FUNCTION_BLOCK fb_debugData
VAR_INPUT
END_VAR
VAR_OUTPUT
END_VAR
VAR
	productID: INT;
END_VAR

productID := 0;


gvl_param.var_productInfo[productID].name 				:= '---ForDebug---';
gvl_param.var_productInfo[productID].num				:= productID;
gvl_param.var_productInfo[productID].bottomPocketQty 	:= 5;
gvl_param.var_productInfo[productID].vertivalPocketQty 	:= 3;
gvl_param.var_productInfo[productID].startCav 			:= 1;
gvl_param.var_productInfo[productID].cavQty 			:= 8;
gvl_param.var_productInfo[productID].gateLength_max 	:= 30000;
gvl_param.var_productInfo[productID].gateLength_min 	:= 15000;
gvl_param.var_productInfo[productID].pocketSumQty		:= 15;
gvl_param.var_productInfo[productID].autoVels.x.vel		:= 300;
gvl_param.var_productInfo[productID].autoVels.x.acc		:= 10000;
gvl_param.var_productInfo[productID].autoVels.x.dcc		:= 10000;
gvl_param.var_productInfo[productID].autoVels.y.vel		:= 150;
gvl_param.var_productInfo[productID].autoVels.y.acc		:= 10000;
gvl_param.var_productInfo[productID].autoVels.y.dcc		:= 10000;
gvl_param.var_productInfo[productID].autoVels.z.vel		:= 150;
gvl_param.var_productInfo[productID].autoVels.z.acc		:= 10000;
gvl_param.var_productInfo[productID].autoVels.z.dcc		:= 10000;
gvl_param.var_productInfo[productID].manaulVels.x.vel	:= 100;
gvl_param.var_productInfo[productID].manaulVels.y.vel	:= 50;
gvl_param.var_productInfo[productID].manaulVels.z.vel	:= 50;

gvl_param.var_productInfo[productID].teachPos.initial.x	:= 950;
gvl_param.var_productInfo[productID].teachPos.initial.y	:= 30;
gvl_param.var_productInfo[productID].teachPos.initial.z	:= 0;
gvl_param.var_productInfo[productID].teachPos.pickUp.x	:= 1250;
gvl_param.var_productInfo[productID].teachPos.pickUp.y	:= 30;
gvl_param.var_productInfo[productID].teachPos.pickUp.z	:= 10;
gvl_param.var_productInfo[productID].teachPos.remove.x	:= 1220;
gvl_param.var_productInfo[productID].teachPos.remove.y	:= 190;
gvl_param.var_productInfo[productID].teachPos.remove.z	:= 10;
//#1
gvl_param.var_productInfo[productID].teachPos.palletize.upperLower[1].cav[1].Pos[1].x := 1007;
gvl_param.var_productInfo[productID].teachPos.palletize.upperLower[1].cav[1].Pos[1].y := 54;
gvl_param.var_productInfo[productID].teachPos.palletize.upperLower[1].cav[1].Pos[1].z := 15;
gvl_param.var_productInfo[productID].teachPos.palletize.upperLower[1].cav[1].Pos[2].x := 1084;
gvl_param.var_productInfo[productID].teachPos.palletize.upperLower[1].cav[1].Pos[2].y := 54;
gvl_param.var_productInfo[productID].teachPos.palletize.upperLower[1].cav[1].Pos[2].z := 15;
gvl_param.var_productInfo[productID].teachPos.palletize.upperLower[1].cav[1].Pos[3].x := 1007;
gvl_param.var_productInfo[productID].teachPos.palletize.upperLower[1].cav[1].Pos[3].y := 256;
gvl_param.var_productInfo[productID].teachPos.palletize.upperLower[1].cav[1].Pos[3].z := 15;
gvl_param.var_productInfo[productID].teachPos.palletize.upperLower[2].cav[1].Pos[1].x := 1007;
gvl_param.var_productInfo[productID].teachPos.palletize.upperLower[2].cav[1].Pos[1].y := 54;
gvl_param.var_productInfo[productID].teachPos.palletize.upperLower[2].cav[1].Pos[1].z := 30;
gvl_param.var_productInfo[productID].teachPos.palletize.upperLower[2].cav[1].Pos[2].x := 1084;
gvl_param.var_productInfo[productID].teachPos.palletize.upperLower[2].cav[1].Pos[2].y := 54;
gvl_param.var_productInfo[productID].teachPos.palletize.upperLower[2].cav[1].Pos[2].z := 30;
gvl_param.var_productInfo[productID].teachPos.palletize.upperLower[2].cav[1].Pos[3].x := 1007;
gvl_param.var_productInfo[productID].teachPos.palletize.upperLower[2].cav[1].Pos[3].y := 256;
gvl_param.var_productInfo[productID].teachPos.palletize.upperLower[2].cav[1].Pos[3].z := 30;
//#2
gvl_param.var_productInfo[productID].teachPos.palletize.upperLower[1].cav[2].Pos[1].x := 886;
gvl_param.var_productInfo[productID].teachPos.palletize.upperLower[1].cav[2].Pos[1].y := 54;
gvl_param.var_productInfo[productID].teachPos.palletize.upperLower[1].cav[2].Pos[1].z := 15;
gvl_param.var_productInfo[productID].teachPos.palletize.upperLower[1].cav[2].Pos[2].x := 963;
gvl_param.var_productInfo[productID].teachPos.palletize.upperLower[1].cav[2].Pos[2].y := 54;
gvl_param.var_productInfo[productID].teachPos.palletize.upperLower[1].cav[2].Pos[2].z := 15;
gvl_param.var_productInfo[productID].teachPos.palletize.upperLower[1].cav[2].Pos[3].x := 886;
gvl_param.var_productInfo[productID].teachPos.palletize.upperLower[1].cav[2].Pos[3].y := 256;
gvl_param.var_productInfo[productID].teachPos.palletize.upperLower[1].cav[2].Pos[3].z := 15;
gvl_param.var_productInfo[productID].teachPos.palletize.upperLower[2].cav[2].Pos[1].x := 886;
gvl_param.var_productInfo[productID].teachPos.palletize.upperLower[2].cav[2].Pos[1].y := 54;
gvl_param.var_productInfo[productID].teachPos.palletize.upperLower[2].cav[2].Pos[1].z := 30;
gvl_param.var_productInfo[productID].teachPos.palletize.upperLower[2].cav[2].Pos[2].x := 963;
gvl_param.var_productInfo[productID].teachPos.palletize.upperLower[2].cav[2].Pos[2].y := 54;
gvl_param.var_productInfo[productID].teachPos.palletize.upperLower[2].cav[2].Pos[2].z := 30;
gvl_param.var_productInfo[productID].teachPos.palletize.upperLower[2].cav[2].Pos[3].x := 886;
gvl_param.var_productInfo[productID].teachPos.palletize.upperLower[2].cav[2].Pos[3].y := 256;
gvl_param.var_productInfo[productID].teachPos.palletize.upperLower[2].cav[2].Pos[3].z := 30;
//#3
gvl_param.var_productInfo[productID].teachPos.palletize.upperLower[1].cav[3].Pos[1].x := 706;
gvl_param.var_productInfo[productID].teachPos.palletize.upperLower[1].cav[3].Pos[1].y := 54;
gvl_param.var_productInfo[productID].teachPos.palletize.upperLower[1].cav[3].Pos[1].z := 15;
gvl_param.var_productInfo[productID].teachPos.palletize.upperLower[1].cav[3].Pos[2].x := 784;
gvl_param.var_productInfo[productID].teachPos.palletize.upperLower[1].cav[3].Pos[2].y := 54;
gvl_param.var_productInfo[productID].teachPos.palletize.upperLower[1].cav[3].Pos[2].z := 15;
gvl_param.var_productInfo[productID].teachPos.palletize.upperLower[1].cav[3].Pos[3].x := 706;
gvl_param.var_productInfo[productID].teachPos.palletize.upperLower[1].cav[3].Pos[3].y := 256;
gvl_param.var_productInfo[productID].teachPos.palletize.upperLower[1].cav[3].Pos[3].z := 15;
gvl_param.var_productInfo[productID].teachPos.palletize.upperLower[2].cav[3].Pos[1].x := 706;
gvl_param.var_productInfo[productID].teachPos.palletize.upperLower[2].cav[3].Pos[1].y := 54;
gvl_param.var_productInfo[productID].teachPos.palletize.upperLower[2].cav[3].Pos[1].z := 30;
gvl_param.var_productInfo[productID].teachPos.palletize.upperLower[2].cav[3].Pos[2].x := 783;
gvl_param.var_productInfo[productID].teachPos.palletize.upperLower[2].cav[3].Pos[2].y := 54;
gvl_param.var_productInfo[productID].teachPos.palletize.upperLower[2].cav[3].Pos[2].z := 30;
gvl_param.var_productInfo[productID].teachPos.palletize.upperLower[2].cav[3].Pos[3].x := 706;
gvl_param.var_productInfo[productID].teachPos.palletize.upperLower[2].cav[3].Pos[3].y := 256;
gvl_param.var_productInfo[productID].teachPos.palletize.upperLower[2].cav[3].Pos[3].z := 30;
//#4
gvl_param.var_productInfo[productID].teachPos.palletize.upperLower[1].cav[4].Pos[1].x := 585;
gvl_param.var_productInfo[productID].teachPos.palletize.upperLower[1].cav[4].Pos[1].y := 54;
gvl_param.var_productInfo[productID].teachPos.palletize.upperLower[1].cav[4].Pos[1].z := 15;
gvl_param.var_productInfo[productID].teachPos.palletize.upperLower[1].cav[4].Pos[2].x := 662;
gvl_param.var_productInfo[productID].teachPos.palletize.upperLower[1].cav[4].Pos[2].y := 54;
gvl_param.var_productInfo[productID].teachPos.palletize.upperLower[1].cav[4].Pos[2].z := 15;
gvl_param.var_productInfo[productID].teachPos.palletize.upperLower[1].cav[4].Pos[3].x := 585;
gvl_param.var_productInfo[productID].teachPos.palletize.upperLower[1].cav[4].Pos[3].y := 256;
gvl_param.var_productInfo[productID].teachPos.palletize.upperLower[1].cav[4].Pos[3].z := 15;
gvl_param.var_productInfo[productID].teachPos.palletize.upperLower[2].cav[4].Pos[1].x := 585;
gvl_param.var_productInfo[productID].teachPos.palletize.upperLower[2].cav[4].Pos[1].y := 54;
gvl_param.var_productInfo[productID].teachPos.palletize.upperLower[2].cav[4].Pos[1].z := 30;
gvl_param.var_productInfo[productID].teachPos.palletize.upperLower[2].cav[4].Pos[2].x := 663;
gvl_param.var_productInfo[productID].teachPos.palletize.upperLower[2].cav[4].Pos[2].y := 54;
gvl_param.var_productInfo[productID].teachPos.palletize.upperLower[2].cav[4].Pos[2].z := 30;
gvl_param.var_productInfo[productID].teachPos.palletize.upperLower[2].cav[4].Pos[3].x := 585;
gvl_param.var_productInfo[productID].teachPos.palletize.upperLower[2].cav[4].Pos[3].y := 256;
gvl_param.var_productInfo[productID].teachPos.palletize.upperLower[2].cav[4].Pos[3].z := 30;
//#5
gvl_param.var_productInfo[productID].teachPos.palletize.upperLower[1].cav[5].Pos[1].x := 406;
gvl_param.var_productInfo[productID].teachPos.palletize.upperLower[1].cav[5].Pos[1].y := 54;
gvl_param.var_productInfo[productID].teachPos.palletize.upperLower[1].cav[5].Pos[1].z := 15;
gvl_param.var_productInfo[productID].teachPos.palletize.upperLower[1].cav[5].Pos[2].x := 484;
gvl_param.var_productInfo[productID].teachPos.palletize.upperLower[1].cav[5].Pos[2].y := 54;
gvl_param.var_productInfo[productID].teachPos.palletize.upperLower[1].cav[5].Pos[2].z := 15;
gvl_param.var_productInfo[productID].teachPos.palletize.upperLower[1].cav[5].Pos[3].x := 406;
gvl_param.var_productInfo[productID].teachPos.palletize.upperLower[1].cav[5].Pos[3].y := 256;
gvl_param.var_productInfo[productID].teachPos.palletize.upperLower[1].cav[5].Pos[3].z := 15;
gvl_param.var_productInfo[productID].teachPos.palletize.upperLower[2].cav[5].Pos[1].x := 405;
gvl_param.var_productInfo[productID].teachPos.palletize.upperLower[2].cav[5].Pos[1].y := 54;
gvl_param.var_productInfo[productID].teachPos.palletize.upperLower[2].cav[5].Pos[1].z := 30;
gvl_param.var_productInfo[productID].teachPos.palletize.upperLower[2].cav[5].Pos[2].x := 483;
gvl_param.var_productInfo[productID].teachPos.palletize.upperLower[2].cav[5].Pos[2].y := 54;
gvl_param.var_productInfo[productID].teachPos.palletize.upperLower[2].cav[5].Pos[2].z := 30;
gvl_param.var_productInfo[productID].teachPos.palletize.upperLower[2].cav[5].Pos[3].x := 405;
gvl_param.var_productInfo[productID].teachPos.palletize.upperLower[2].cav[5].Pos[3].y := 256;
gvl_param.var_productInfo[productID].teachPos.palletize.upperLower[2].cav[5].Pos[3].z := 30;
//#6
gvl_param.var_productInfo[productID].teachPos.palletize.upperLower[1].cav[6].Pos[1].x := 286;
gvl_param.var_productInfo[productID].teachPos.palletize.upperLower[1].cav[6].Pos[1].y := 54;
gvl_param.var_productInfo[productID].teachPos.palletize.upperLower[1].cav[6].Pos[1].z := 15;
gvl_param.var_productInfo[productID].teachPos.palletize.upperLower[1].cav[6].Pos[2].x := 363;
gvl_param.var_productInfo[productID].teachPos.palletize.upperLower[1].cav[6].Pos[2].y := 54;
gvl_param.var_productInfo[productID].teachPos.palletize.upperLower[1].cav[6].Pos[2].z := 15;
gvl_param.var_productInfo[productID].teachPos.palletize.upperLower[1].cav[6].Pos[3].x := 286;
gvl_param.var_productInfo[productID].teachPos.palletize.upperLower[1].cav[6].Pos[3].y := 256;
gvl_param.var_productInfo[productID].teachPos.palletize.upperLower[1].cav[6].Pos[3].z := 15;
gvl_param.var_productInfo[productID].teachPos.palletize.upperLower[2].cav[6].Pos[1].x := 285;
gvl_param.var_productInfo[productID].teachPos.palletize.upperLower[2].cav[6].Pos[1].y := 54;
gvl_param.var_productInfo[productID].teachPos.palletize.upperLower[2].cav[6].Pos[1].z := 30;
gvl_param.var_productInfo[productID].teachPos.palletize.upperLower[2].cav[6].Pos[2].x := 362;
gvl_param.var_productInfo[productID].teachPos.palletize.upperLower[2].cav[6].Pos[2].y := 54;
gvl_param.var_productInfo[productID].teachPos.palletize.upperLower[2].cav[6].Pos[2].z := 30;
gvl_param.var_productInfo[productID].teachPos.palletize.upperLower[2].cav[6].Pos[3].x := 285;
gvl_param.var_productInfo[productID].teachPos.palletize.upperLower[2].cav[6].Pos[3].y := 256;
gvl_param.var_productInfo[productID].teachPos.palletize.upperLower[2].cav[6].Pos[3].z := 30;
//#7
gvl_param.var_productInfo[productID].teachPos.palletize.upperLower[1].cav[7].Pos[1].x := 107;
gvl_param.var_productInfo[productID].teachPos.palletize.upperLower[1].cav[7].Pos[1].y := 54;
gvl_param.var_productInfo[productID].teachPos.palletize.upperLower[1].cav[7].Pos[1].z := 15;
gvl_param.var_productInfo[productID].teachPos.palletize.upperLower[1].cav[7].Pos[2].x := 184;
gvl_param.var_productInfo[productID].teachPos.palletize.upperLower[1].cav[7].Pos[2].y := 54;
gvl_param.var_productInfo[productID].teachPos.palletize.upperLower[1].cav[7].Pos[2].z := 15;
gvl_param.var_productInfo[productID].teachPos.palletize.upperLower[1].cav[7].Pos[3].x := 107;
gvl_param.var_productInfo[productID].teachPos.palletize.upperLower[1].cav[7].Pos[3].y := 256;
gvl_param.var_productInfo[productID].teachPos.palletize.upperLower[1].cav[7].Pos[3].z := 15;
gvl_param.var_productInfo[productID].teachPos.palletize.upperLower[2].cav[7].Pos[1].x := 106;
gvl_param.var_productInfo[productID].teachPos.palletize.upperLower[2].cav[7].Pos[1].y := 54;
gvl_param.var_productInfo[productID].teachPos.palletize.upperLower[2].cav[7].Pos[1].z := 30;
gvl_param.var_productInfo[productID].teachPos.palletize.upperLower[2].cav[7].Pos[2].x := 183;
gvl_param.var_productInfo[productID].teachPos.palletize.upperLower[2].cav[7].Pos[2].y := 54;
gvl_param.var_productInfo[productID].teachPos.palletize.upperLower[2].cav[7].Pos[2].z := 30;
gvl_param.var_productInfo[productID].teachPos.palletize.upperLower[2].cav[7].Pos[3].x := 106;
gvl_param.var_productInfo[productID].teachPos.palletize.upperLower[2].cav[7].Pos[3].y := 256;
gvl_param.var_productInfo[productID].teachPos.palletize.upperLower[2].cav[7].Pos[3].z := 30;
//#8
gvl_param.var_productInfo[productID].teachPos.palletize.upperLower[1].cav[8].Pos[1].x := -13;
gvl_param.var_productInfo[productID].teachPos.palletize.upperLower[1].cav[8].Pos[1].y := 54;
gvl_param.var_productInfo[productID].teachPos.palletize.upperLower[1].cav[8].Pos[1].z := 15;
gvl_param.var_productInfo[productID].teachPos.palletize.upperLower[1].cav[8].Pos[2].x := 63;
gvl_param.var_productInfo[productID].teachPos.palletize.upperLower[1].cav[8].Pos[2].y := 54;
gvl_param.var_productInfo[productID].teachPos.palletize.upperLower[1].cav[8].Pos[2].z := 15;
gvl_param.var_productInfo[productID].teachPos.palletize.upperLower[1].cav[8].Pos[3].x := -13;
gvl_param.var_productInfo[productID].teachPos.palletize.upperLower[1].cav[8].Pos[3].y := 256;
gvl_param.var_productInfo[productID].teachPos.palletize.upperLower[1].cav[8].Pos[3].z := 15;
gvl_param.var_productInfo[productID].teachPos.palletize.upperLower[2].cav[8].Pos[1].x := -14;
gvl_param.var_productInfo[productID].teachPos.palletize.upperLower[2].cav[8].Pos[1].y := 54;
gvl_param.var_productInfo[productID].teachPos.palletize.upperLower[2].cav[8].Pos[1].z := 30;
gvl_param.var_productInfo[productID].teachPos.palletize.upperLower[2].cav[8].Pos[2].x := 62;
gvl_param.var_productInfo[productID].teachPos.palletize.upperLower[2].cav[8].Pos[2].y := 54;
gvl_param.var_productInfo[productID].teachPos.palletize.upperLower[2].cav[8].Pos[2].z := 30;
gvl_param.var_productInfo[productID].teachPos.palletize.upperLower[2].cav[8].Pos[3].x := -14;
gvl_param.var_productInfo[productID].teachPos.palletize.upperLower[2].cav[8].Pos[3].y := 256;
gvl_param.var_productInfo[productID].teachPos.palletize.upperLower[2].cav[8].Pos[3].z := 30;

//sample
gvl_param.var_productInfo[productID].teachPos.sample[1].x := 1263;
gvl_param.var_productInfo[productID].teachPos.sample[1].y := 296;
gvl_param.var_productInfo[productID].teachPos.sample[1].z := 10;
gvl_param.var_productInfo[productID].teachPos.sample[2].x := 1242;
gvl_param.var_productInfo[productID].teachPos.sample[2].y := 296;
gvl_param.var_productInfo[productID].teachPos.sample[2].z := 10;
gvl_param.var_productInfo[productID].teachPos.sample[3].x := 1222;
gvl_param.var_productInfo[productID].teachPos.sample[3].y := 296;
gvl_param.var_productInfo[productID].teachPos.sample[3].z := 10;
gvl_param.var_productInfo[productID].teachPos.sample[4].x := 1202;
gvl_param.var_productInfo[productID].teachPos.sample[4].y := 296;
gvl_param.var_productInfo[productID].teachPos.sample[4].z := 10;
gvl_param.var_productInfo[productID].teachPos.sample[5].x := 1262;
gvl_param.var_productInfo[productID].teachPos.sample[5].y := 187;
gvl_param.var_productInfo[productID].teachPos.sample[5].z := 10;
gvl_param.var_productInfo[productID].teachPos.sample[6].x := 1242;
gvl_param.var_productInfo[productID].teachPos.sample[6].y := 187;
gvl_param.var_productInfo[productID].teachPos.sample[6].z := 10;
gvl_param.var_productInfo[productID].teachPos.sample[7].x := 1222;
gvl_param.var_productInfo[productID].teachPos.sample[7].y := 187;
gvl_param.var_productInfo[productID].teachPos.sample[7].z := 10;
gvl_param.var_productInfo[productID].teachPos.sample[8].x := 1202;
gvl_param.var_productInfo[productID].teachPos.sample[8].y := 187;
gvl_param.var_productInfo[productID].teachPos.sample[8].z := 10;

END_FUNCTION_BLOCK

(* stored: Version 1.1.0.1, ProductVersion 3.1.4024.11
   POU fb_debugData: Id {0311ba4b-b359-482f-a223-abfe5fe63057}, SpecialFunc None *)
